Universal Robots PolyScope program: interconnect.urp

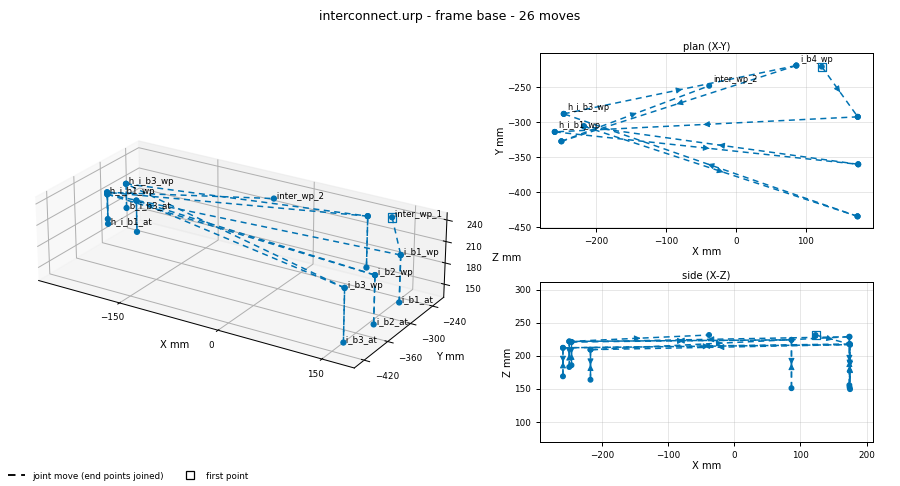
[picture p0: tool path of interconnect.urp in frame base, 26 of 26 moves have a stored position in this frame; points joined in program order, loops and branches not executed]
Program interconnect (installation=default directory=/programs/Session 1 createdIn=5.3.1.64192 lastSavedIn=5.3.1.64192 robotSerialNumber=20195300365)
Calibrated DH parameters: a=[-0.000093, -0.190649, -0.212673, 0.000091, -0.000205, 0]; d=[0.151591, 44.061648, -42.488068, -1.442789, 0.085322, 0.091911]; alpha=[1.570082, -0.003447, 0.007513, 1.572293, -1.571904, 0]; deltaTheta=[0, -0.672656, 0.728185, -0.055522, 0.000005, 0]
Robot Program (runOnlyOnce=true)
  URCap Gripper Activate (Robotiq_Grippers, Robotiq Inc.) dataModel(ResetAndActivateKey=false)
  URCap Gripper (Robotiq_Grippers, Robotiq Inc.) dataModel(position=50.0, force=100.0, speed=100.0, positionInDouble=50.0, forceInDouble=100.0, speedInDouble=100.0, slaveIds=[9], blocking=true)
  MoveJ speed 60 deg/s, acceleration 80 deg/s^2 (useActiveTCP=true) feature=Base
    Waypoint inter_wp_1: TCP in base x=122.78 y=-220.583 z=231.495 mm, rx=2.2968 ry=2.1205 rz=-0.0201 rad; joints [-29.631, -72.124, -124.848, -72.343, 89.412, -204.687] deg
  Folder Interconnect
    MoveJ speed 60 deg/s, acceleration 80 deg/s^2 (useActiveTCP=true) feature=Base
      Waypoint i_b1_wp: TCP in base x=174.192 y=-292.235 z=217.966 mm, rx=2.2497 ry=2.1639 rz=-0.0066 rad; joints [-36.697, -97.49, -106.294, -65.059, 89.868, -214.094] deg
      Waypoint i_b1_at: TCP in base x=174.179 y=-292.238 z=152.33 mm, rx=2.2498 ry=2.1638 rz=-0.0066 rad; joints [-36.724, -106.455, -115.875, -46.513, 89.778, -214.022] deg
      URCap Gripper (Robotiq_Grippers, Robotiq Inc.) dataModel(position=100.0, force=100.0, speed=100.0, positionInDouble=100.0, forceInDouble=100.0, speedInDouble=100.0, slaveIds=[9], blocking=true)
      Waypoint i_b1_wp: TCP in base x=174.192 y=-292.235 z=217.966 mm, rx=2.2497 ry=2.1639 rz=-0.0066 rad; joints [-36.697, -97.49, -106.294, -65.059, 89.868, -214.094] deg
      Waypoint h_i_b1_wp: TCP in base x=-258.783 y=-313.738 z=212.193 mm, rx=-3.0753 ry=0.0547 rz=-0.0056 rad; joints [-110.639, -114.762, -82.85, -75.951, 89.224, -198.304] deg
      Waypoint h_i_b1_at: TCP in base x=-258.784 y=-313.742 z=169.111 mm, rx=-3.0753 ry=0.0547 rz=-0.0057 rad; joints [-110.657, -118.67, -89.325, -65.57, 89.197, -198.259] deg
      URCap Gripper (Robotiq_Grippers, Robotiq Inc.) dataModel(position=50.0, force=100.0, speed=100.0, positionInDouble=50.0, forceInDouble=100.0, speedInDouble=100.0, slaveIds=[9], blocking=true)
      Waypoint h_i_b1_wp: TCP in base x=-258.783 y=-313.738 z=212.193 mm, rx=-3.0753 ry=0.0547 rz=-0.0056 rad; joints [-110.639, -114.762, -82.85, -75.951, 89.224, -198.304] deg
    MoveJ speed 60 deg/s, acceleration 80 deg/s^2 (useActiveTCP=true) feature=Base
      Waypoint i_b2_wp: TCP in base x=174.829 y=-360.086 z=217.004 mm, rx=2.2647 ry=2.1469 rz=-0.0178 rad; joints [-45.021, -111.703, -87.984, -69.069, 89.592, -221.659] deg
      Waypoint i_b2_at: TCP in base x=174.839 y=-360.085 z=149.76 mm, rx=2.2646 ry=2.147 rz=-0.0179 rad; joints [-45.043, -119.061, -97.021, -52.674, 89.527, -221.597] deg
      URCap Gripper (Robotiq_Grippers, Robotiq Inc.) dataModel(position=100.0, force=100.0, speed=100.0, positionInDouble=100.0, forceInDouble=100.0, speedInDouble=100.0, slaveIds=[9], blocking=true)
      Waypoint i_b2_wp: TCP in base x=174.829 y=-360.086 z=217.004 mm, rx=2.2647 ry=2.1469 rz=-0.0178 rad; joints [-45.021, -111.703, -87.984, -69.069, 89.592, -221.659] deg
      Waypoint h_i_b2_wp: TCP in base x=-217.209 y=-305.752 z=209.413 mm, rx=-3.1147 ry=0.0762 rz=0.0244 rad; joints [-104.846, -106.933, -95.847, -68.393, 89.071, -191.695] deg
      Waypoint h_i_b2_at: TCP in base x=-217.212 y=-305.747 z=163.983 mm, rx=-3.1147 ry=0.0762 rz=0.0244 rad; joints [-104.864, -112.08, -102.369, -56.726, 89.025, -191.646] deg
      URCap Gripper (Robotiq_Grippers, Robotiq Inc.) dataModel(position=50.0, force=100.0, speed=100.0, positionInDouble=50.0, forceInDouble=100.0, speedInDouble=100.0, slaveIds=[9], blocking=true)
      Waypoint h_i_b2_wp: TCP in base x=-217.209 y=-305.752 z=209.413 mm, rx=-3.1147 ry=0.0762 rz=0.0244 rad; joints [-104.846, -106.933, -95.847, -68.393, 89.071, -191.695] deg
    MoveJ speed 60 deg/s, acceleration 80 deg/s^2 (useActiveTCP=true) feature=Base
      Waypoint i_b3_wp: TCP in base x=173.862 y=-434.439 z=228.912 mm, rx=-2.2984 ry=-2.1342 rz=0.0077 rad; joints [-51.956, -128.706, -57.062, -84.438, 89.974, -227.564] deg
      Waypoint i_b3_at: TCP in base x=173.823 y=-434.448 z=155.772 mm, rx=-2.2985 ry=-2.1341 rz=0.0077 rad; joints [-51.993, -133.364, -69.125, -67.717, 89.949, -227.489] deg
      URCap Gripper (Robotiq_Grippers, Robotiq Inc.) dataModel(position=100.0, force=100.0, speed=100.0, positionInDouble=100.0, forceInDouble=100.0, speedInDouble=100.0, slaveIds=[9], blocking=true)
      Waypoint i_b3_wp: TCP in base x=173.862 y=-434.439 z=228.912 mm, rx=-2.2984 ry=-2.1342 rz=0.0077 rad; joints [-51.956, -128.706, -57.062, -84.438, 89.974, -227.564] deg
      Waypoint h_i_b3_wp: TCP in base x=-245.926 y=-287.976 z=221.138 mm, rx=2.2651 ry=2.1423 rz=0.0503 rad; joints [-110.984, -107.188, -92.208, -71.613, 92.308, -287.496] deg
      Waypoint b_i_b3_at: TCP in base x=-245.92 y=-287.99 z=185.909 mm, rx=2.265 ry=2.1423 rz=0.0502 rad; joints [-110.998, -110.532, -97.867, -62.605, 92.28, -287.458] deg
      URCap Gripper (Robotiq_Grippers, Robotiq Inc.) dataModel(position=50.0, force=100.0, speed=100.0, positionInDouble=50.0, forceInDouble=100.0, speedInDouble=100.0, slaveIds=[9], blocking=true)
      Waypoint h_i_b3_wp: TCP in base x=-245.926 y=-287.976 z=221.138 mm, rx=2.2651 ry=2.1423 rz=0.0503 rad; joints [-110.984, -107.188, -92.208, -71.613, 92.308, -287.496] deg
    MoveJ speed 60 deg/s, acceleration 80 deg/s^2 (useActiveTCP=true) feature=Base
      Waypoint i_b4_wp: TCP in base x=86.376 y=-218.928 z=224.266 mm, rx=2.2427 ry=2.1745 rz=0.0062 rad; joints [-35.112, -67.186, -129.953, -71.753, 90.433, -212.954] deg
      Waypoint i_b4_at: TCP in base x=86.374 y=-218.929 z=151.179 mm, rx=2.2427 ry=2.1745 rz=0.0061 rad; joints [-35.159, -80.22, -144.952, -43.721, 90.288, -212.837] deg
      URCap Gripper (Robotiq_Grippers, Robotiq Inc.) dataModel(position=100.0, force=100.0, speed=100.0, positionInDouble=100.0, forceInDouble=100.0, speedInDouble=100.0, slaveIds=[9], blocking=true)
      Waypoint i_b4_wp: TCP in base x=86.376 y=-218.928 z=224.266 mm, rx=2.2427 ry=2.1745 rz=0.0062 rad; joints [-35.112, -67.186, -129.953, -71.753, 90.433, -212.954] deg
      Waypoint h_i_b4_wp: TCP in base x=-249.299 y=-327.199 z=221.841 mm, rx=2.2374 ry=2.2006 rz=0.0433 rad; joints [-109.1, -114.821, -80.967, -75.483, 91.148, -287.896] deg
      Waypoint h_i_b4_at: TCP in base x=-249.283 y=-327.216 z=183.232 mm, rx=2.2374 ry=2.2006 rz=0.0433 rad; joints [-109.114, -117.988, -87.16, -66.124, 91.124, -287.854] deg
      URCap Gripper (Robotiq_Grippers, Robotiq Inc.) dataModel(position=50.0, force=100.0, speed=100.0, positionInDouble=50.0, forceInDouble=100.0, speedInDouble=100.0, slaveIds=[9], blocking=true)
      Waypoint h_i_b4_wp: TCP in base x=-249.299 y=-327.199 z=221.841 mm, rx=2.2374 ry=2.2006 rz=0.0433 rad; joints [-109.1, -114.821, -80.967, -75.483, 91.148, -287.896] deg
  MoveJ speed 60 deg/s, acceleration 80 deg/s^2 (useActiveTCP=true) feature=Base
    Waypoint inter_wp_2: TCP in base x=-38.107 y=-247.898 z=231.572 mm, rx=2.241 ry=2.1798 rz=0.019 rad; joints [-68.076, -72.135, -124.793, -72.457, 91.361, -246.109] deg
